PROGRAM MAIN
VAR
	Timer1 :TON;
	Timer2 : TON;
	PulseTimer1 : TP;

	CurrentState  : States;
	
	ServoRTrigY : R_Trig ; 
	ServoRTrigX : R_Trig ; 
	
	//Eigen trigger booleans
	InitYReady : BOOL;
	InitXReady : BOOL;

	Test : Moving;
	Pos : INT;
	ActualPos : int;
END_VAR

PulseTimer1(IN:=GVL_IO.Start_button, PT:=T#150MS);

Timer1(IN:= GVL_IO.a_1_Vertical_Zaxis_downward, PT:= T#10MS);

CASE CurrentState OF
States.Init:
		//Aanzetten van servo's. Dit kan even duren GEEN HOMING
		GVL_IO.SVONX_SERVO_ON_tableX 	  := TRUE; 
		GVL_IO.SVONY_SERVO_ON_translY 	  := TRUE;
		
		GVL_IO.SETUPX_ORIGIN_tableX := PulseTimer1.Q;
		GVL_IO.SETUPY_ORIGIN_translY := PulseTimer1.Q;
		
		//// Koppelen van outputs Busy aan var's. Triggered op een falling edge.
		IF PulseTimer1.Q THEN
			ServoRTrigX ( clk := gvl_io.SETONX_ORIGIN_tableX ); 
	  		ServoRTrigY ( clk := gvl_io.SETONY_ORIGIN_translationY );
		END_IF
		
		// Bools setten aan de hand van triggers.
		IF ServoRTrigX.Q THEN
			InitXReady:= TRUE;
		END_IF
		
		IF ServoRTrigY.Q THEN
			InitYReady:= TRUE;
		END_IF
		
		// Init voltooid ga naar idle
		IF InitXReady AND InitYReady THEN
			Pos:= 1;
			ActualPos:= 0;
			CurrentState:= States.Idle;
		END_IF
		
States.Idle:
		IF NOT GVL_IO.Stop_button AND NOT GVL_IO.dp2_Cover_detection THEN
			//SEND MESSAGEE TODO
			CurrentState := States.Idle;
		END_IF
		
		IF NOT GVL_IO.Stop_button AND GVL_IO.dp1_Can_detection AND GVL_IO.dp2_Cover_detection THEN
			CurrentState := States.MoveToPickUp; //TODO stopbutton
		END_IF
		
		IF Pos >= 26 THEN
			CurrentState := States.PalletFull;
		END_IF
		
States.MoveToPickUp:

		Test(Position:=0);
		IF NOT Test.Busy THEN
			CurrentState := States.PickUpDown;
		END_IF
		
		
States.PickUpDown:
		IF GVL_IO.a_0_Vertical_Zaxis_upward THEN
			GVL_IO.Aplus_Vert_axis_downwards := TRUE;
		END_IF
		
		IF GVL_IO.a_1_Vertical_Zaxis_downward THEN
			GVL_IO.Vplus_Vacuum_start := TRUE;
			
			IF Timer1.Q THEN
			CurrentState := States.PickUpUp;
			END_IF
		END_IF

States.PickUpUp:
		GVL_IO.Aplus_Vert_axis_downwards := FALSE;
		
		IF GVL_IO.a_0_Vertical_Zaxis_upward THEN
			CurrentState := States.Moving;
		END_IF
		
States.Moving:
		Test(Position:=Pos);
		IF NOT Test.Busy THEN
			Pos:= Pos + 1;
			ActualPos:= ActualPos + 1;
			CurrentState := States.DropDown;
		END_IF
		
States.DropDown:
		IF GVL_IO.a_0_Vertical_Zaxis_upward THEN
			GVL_IO.Aplus_Vert_axis_downwards := TRUE;
		END_IF
		
		IF 	GVL_IO.a_1_Vertical_Zaxis_downward THEN
			GVL_IO.Vplus_Vacuum_start := FALSE;
			Timer2(IN:=GVL_IO.a_1_Vertical_Zaxis_downward, PT:=T#10MS);
			IF Timer2.Q THEN
				CurrentState := States.DropUp;
			END_IF
		END_IF


States.DropUp:
		IF GVL_IO.a_1_Vertical_Zaxis_downward THEN
			GVL_IO.Aplus_Vert_axis_downwards := FALSE;
		END_IF
		
		IF GVL_IO.a_0_Vertical_Zaxis_upward THEN
			CurrentState := States.Idle;
		END_IF
		
States.PalletFull:
		GVL_IO.BR_Alarm_light := TRUE;
		IF GVL_IO.Reset_button THEN
			GVL_IO.BR_Alarm_light := FALSE;
			Pos := 1;
			ActualPos := 0;
			Currentstate := States.Idle;
		END_IF
END_CASE

END_PROGRAM

(* stored: Version 1.1.0.1, ProductVersion 3.1.4022.12
   POU MAIN: Id {a4f99ad4-3d99-4cc3-aec6-4b8f25d45e95}, SpecialFunc None *)
